// SIMATIC S7-200 project (STEP 7-Micro/WIN), CPU 224XP REL 02.01

SYMBOL_TABLE USER1
S_tar            I0.0
S_top            I0.1
Trung_gian       M0.0
Muc_be_tren      I0.2
Bom_1            Q0.0
Bom_2            Q0.1
END_SYMBOL_TABLE

ORGANIZATION_BLOCK MAIN:OB1
TITLE=PROGRAM COMMENTS
BEGIN
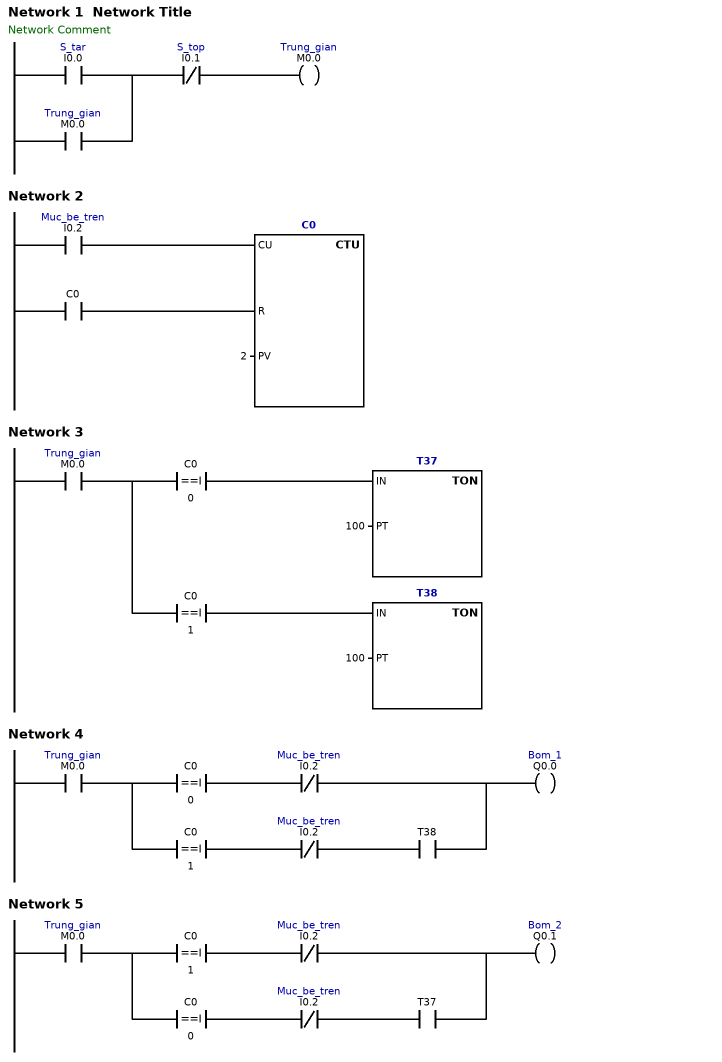
Network 1 // Network Title
// Network Comment
LD     S_tar:I0.0
O      Trung_gian:M0.0
AN     S_top:I0.1
=      Trung_gian:M0.0
Network 2
LD     Muc_be_tren:I0.2
LD     C0
CTU    C0, 2
Network 3
LD     Trung_gian:M0.0
LPS
AW=    C0, 0
TON    T37, 100
LPP
AW=    C0, 1
TON    T38, 100
Network 4
LD     Trung_gian:M0.0
LDW=   C0, 0
AN     Muc_be_tren:I0.2
LDW=   C0, 1
AN     Muc_be_tren:I0.2
A      T38
OLD
ALD
=      Bom_1:Q0.0
Network 5
LD     Trung_gian:M0.0
LDW=   C0, 1
AN     Muc_be_tren:I0.2
LDW=   C0, 0
AN     Muc_be_tren:I0.2
A      T37
OLD
ALD
=      Bom_2:Q0.1
END_ORGANIZATION_BLOCK
